{attribute 'qualified_only'}
{attribute 'strict'}
TYPE E_Valve_Error_State :
(
	enum_member := 0
);
END_TYPE

(* stored: Version 1.1.0.1, ProductVersion 3.1.4024.12
   DUT E_Valve_Error_State: Id {eeccb26d-7a85-4e90-93cf-70e7cfcd3abb} *)
